{attribute 'qualified_only'}
{attribute 'strict'}
TYPE E_SequenceList_DM :
(
	SEQ_MAIN := 1,
	SEQ_CALIBRATE := 2,
	SEQ_FILL := 3,
	SEQ_DRAIN := 4
);
END_TYPE

(* stored: Version 1.1.0.1, ProductVersion 3.1.4024.12
   DUT E_SequenceList_DM: Id {a8f12680-3add-4f7e-a79e-59eeb2f898b8} *)
